{attribute 'GeneratedUsingTerminal: EJ6224-0000-0016'}
{attribute addProperty BoxType "EJ6224-0000-0016"}
{attribute addProperty Id "AdsAddrAT %I*AMSADDR8AoeNetIdAT %I*AMSNETID6StateAT %I*UINT2"}
{attribute addProperty CRC "2417512204"}
{attribute addProperty Size "16"}
TYPE InfoData_90184F0C EXTENDS InputBase_8311D824 :
STRUCT
	{attribute addProperty Name "AdsAddr"}
	AdsAddr AT %I* : AMSADDR;
	{attribute addProperty Name "AoeNetId"}
	AoeNetId AT %I* : AMSNETID;
	{attribute addProperty Name "State"}
	State AT %I* : UINT;
END_STRUCT
END_TYPE

(* stored: Version 1.2.0.0, ProductVersion 3.1.4024.11
   DUT InfoData_90184F0C: Id {3a915e7d-f317-47ef-a78b-d4af88b0ed95} *)
